FUNCTION_BLOCK GreenMasterXXL_FB EXTENDS GreenMasterXXL
VAR_INPUT
END_VAR
VAR_OUTPUT
END_VAR
VAR
END_VAR


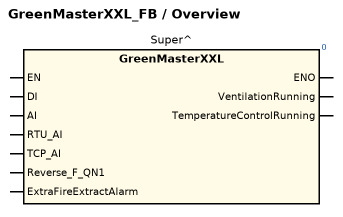
// PAGE Overview
Super^(); // GreenMasterXXL

END_FUNCTION_BLOCK

(* stored: Version 1.1.0.1, ProductVersion 3.1.4024.6
   POU GreenMasterXXL_FB: Id {efde90f3-0b0d-4035-9bd6-c586de412eb2}, SpecialFunc None *)
